Staubli VAL3: SparePoint.pjx

--- SparePoint.pjx ---
Parameters version=s7.8.3 stackSize=5000 millimeterUnit=true
Program file=EditPoint.pgx
Program file=EnterPageKey.pgx
Program file=getPoint.pgx
Program file=Init.pgx
Program file=Main.pgx
Program file=MainKey.pgx
Program file=OnF1.pgx
Program file=OnF2.pgx
Program file=OnF3.pgx
Program file=OnF4.pgx
Program file=OnF5.pgx
Program file=OnF6.pgx
Program file=OnF7.pgx
Program file=OnF8.pgx
Program file=Refresh.pgx
Program file=Refresh2.pgx
Program file=Refresh3.pgx
Program file=RefreshList.pgx
Program file=Save.pgx
Program file=setPoint.pgx
Program file=start.pgx
Program file=stop.pgx
Data file=SparePoint.dtx
Library alias=user path=Disk://userPage/USERPAGE.pjx
Library alias=PublicProg path=Disk://PublicProg/PublicProg.pjx

--- SparePoint.dtx ---
bool bByPass[4]
bool bExit
bool bListRefresh
bool bUserRefresh
frame fFrame = {fatherId=world[0]}
mdesc mNomSpeed
num nPage = 1
num nSelected
public pointRx pPoint{}
  [P1] = {x=495.660657, y=122.165524, z=84.338304, rx=9.53283, ry=179.762496, rz=-66.438432, shoulder=lefty, elbow=epositive, wrist=wpositive, fatherId=world[0]}
  [P10] = {fatherId=world[0]}
  [P11] = {fatherId=world[0]}
  [P12] = {fatherId=world[0]}
  [P13] = {fatherId=world[0]}
  [P14] = {fatherId=world[0]}
  [P15] = {fatherId=world[0]}
  [P16] = {fatherId=world[0]}
  [P2] = {fatherId=world[0]}
  [P3] = {fatherId=world[0]}
  [P4] = {fatherId=world[0]}
  [P5] = {fatherId=world[0]}
  [P6] = {fatherId=world[0]}
  [P7] = {fatherId=world[0]}
  [P8] = {fatherId=world[0]}
  [P9] = {fatherId=world[0]}
public string sDeli[2]
  [0] = "A"
  [1] = "C"
public string sFileList = "A140"
string sFolder = "Disk://Traj/"
string sItem = "P1"
string sList[16]
  [0] = "P1"
  [1] = "P2"
  [2] = "P3"
  [3] = "P4"
  [4] = "P5"
  [5] = "P6"
  [6] = "P7"
  [7] = "P8"
  [8] = "P9"
  [9] = "P10"
  [10] = "P11"
  [11] = "P12"
  [12] = "P13"
  [13] = "P14"
  [14] = "P15"
  [15] = "P16"
string sListItemValue
string sOutputFolder = "Disk://Traj/"
string sParameter
string sPointName = "P1"
string sPtPara

--- Main.pgx ---
program Main()
  local num l_nKey
begin
  //
  do
    call Refresh()
    call RefreshList()
    call user:setList("路径",sList,bUserRefresh,bListRefresh,nSelected,sItem,l_nKey)
    bUserRefresh=false
    bListRefresh=false
    call MainKey(l_nKey)
    delay(0)
  until bExit

end

--- EditPoint.pgx ---
program EditPoint()
  local bool l_bRes
  local num l_i
  local string l_sValue
  local num l_nSelect
  local string l_sItem
  local num l_nKey
  local num l_nRes
begin
//  switch nPage
//    //运动点
//    case 1
//      cls()
//      resize(sParameter,1,11)
//      sParameter[0]="X"
//      sParameter[1]="Y"
//      sParameter[2]="Z"
//      sParameter[3]="Rx"
//      sParameter[4]="Ry"
//      sParameter[5]="Rz"
//      sParameter[6]="P1"
//      sParameter[7]="P2"
//      sParameter[8]="IO1"
//      sParameter[9]="IO2"
//      sParameter[10]="delay"
//      //
//      resize(sListItemValue,1,size(sParameter))
//      sListItemValue[0]=toString(".3",prd:pDemo[nSelected].trsf.x)
//      sListItemValue[1]=toString(".3",prd:pDemo[nSelected].trsf.y)
//      sListItemValue[2]=toString(".3",prd:pDemo[nSelected].trsf.z)
//      sListItemValue[3]=toString(".3",prd:pDemo[nSelected].trsf.rx)
//      sListItemValue[4]=toString(".3",prd:pDemo[nSelected].trsf.ry)
//      sListItemValue[5]=toString(".3",prd:pDemo[nSelected].trsf.rz)
//      //解析sPtParameter
//      call getPtPara(prd:sPtParameter[nSelected],sPtPara)
//      sListItemValue[6]=sPtPara[0]
//      sListItemValue[7]=sPtPara[1]
//      sListItemValue[8]=sPtPara[2]
//      sListItemValue[9]=sPtPara[3]
//      sListItemValue[10]=sPtPara[4]
//      //
//      for l_i=0 to size(sParameter)-1
//        call user:strlength(sParameter[l_i],user:nBottomX/2)
//        l_sValue=sListItemValue[l_i]
//        call user:strlength(l_sValue,user:nBottomX/2+1)
//        sParameter[l_i]=sParameter[l_i]+":"+l_sValue
//      endFor

//      bUserRefresh=true
//      bListRefresh=true
//      //
//      do
//        if bUserRefresh
//          cls()
//          call user:clear(0,13)
//          call user:typeMenu(8,"确定")
//        endIf
//        call user:setList("编辑点",sParameter,bUserRefresh,bListRefresh,l_nSelect,l_sItem,l_nKey)
//        bUserRefresh=false
//        bListRefresh=false
//        call EnterPageKey(l_nKey,l_nSelect,sParameter[l_nSelect])
//        delay(0)
//      until l_nKey==255 or l_nKey==278
//      prd:sPtParameter[nSelected]=sListItemValue[6]+"/"+sListItemValue[7]+"/"+sListItemValue[8]+"/"+sListItemValue[9]+"/"+sListItemValue[10]
//      bUserRefresh=true
//      bListRefresh=true
//    break
//  endSwitch
end

--- EnterPageKey.pgx ---
program EnterPageKey(num& x_nKey, num& x_nSelect, string& x_sItem)
  local string l_sStr
  local num l_nKey
  local string l_sEmpty
  local string l_sValue
  local num l_nItem
  local num l_nView
  local string l_sItem
  local point lp
  local string l_sYN[2]
  local bool l_bRes
  local num l_nTemp
begin
  //
//  //编辑项目
//  switch x_nSelect
//    //X
//    case 0
//      if x_nKey==270
//        call user:editNum(x_sItem,sListItemValue[x_nSelect],prd:pDemo[nSelected].trsf.x,x_nSelect)
//      endIf
//    break
//    //Y
//    case 1
//      if x_nKey==270
//        call user:editNum(x_sItem,sListItemValue[x_nSelect],prd:pDemo[nSelected].trsf.y,x_nSelect)
//      endIf
//    break
//    //Z
//    case 2
//      if x_nKey==270
//        call user:editNum(x_sItem,sListItemValue[x_nSelect],prd:pDemo[nSelected].trsf.z,x_nSelect)
//      endIf
//    break
//    //rx
//    case 3
//      if x_nKey==270
//        call user:editNum(x_sItem,sListItemValue[x_nSelect],prd:pDemo[nSelected].trsf.rx,x_nSelect)
//      endIf
//    break
//    //ry
//    case 4
//      if x_nKey==270
//        call user:editNum(x_sItem,sListItemValue[x_nSelect],prd:pDemo[nSelected].trsf.ry,x_nSelect)
//      endIf
//    break
//    //rz
//    case 5
//      if x_nKey==270
//        call user:editNum(x_sItem,sListItemValue[x_nSelect],prd:pDemo[nSelected].trsf.rz,x_nSelect)
//      endIf
//    break
//    //P1
//    case 6
//      if x_nKey==270
//        // call user:editNum(x_sItem,sListItemValue[x_nSelect],Path:mTrajSpd[nSelectedC].tvel,x_nSelect)
//      endIf
//    break
//    //P2
//    case 7
//      if x_nKey==270
//        //call user:editNum(x_sItem,sListItemValue[x_nSelect],Path:mTrajSpd[nSelectedC].accel,x_nSelect)
//      endIf
//    break
//    //IO1
//    case 8
//      if x_nKey==270
//        call IO:setIO(sListItemValue[x_nSelect])
//        call IO:Main(1)
//        call IO:getIO(sListItemValue[x_nSelect])
//        //
//        x_sItem="IO1      :"+sListItemValue[x_nSelect]
//      endIf

//    break
//    //IO2
//    case 9
//      if x_nKey==270
//        call IO:setIO(sListItemValue[x_nSelect])
//        call IO:Main(1)
//        call IO:getIO(sListItemValue[x_nSelect])
//        //
//        x_sItem="IO2      :"+sListItemValue[x_nSelect]
//      endIf
//    break
//    //delay
//    case 10
//      if x_nKey==270
//        call user:editNum(x_sItem,sListItemValue[x_nSelect],l_nTemp,x_nSelect)
//      endIf
//    break
//  endSwitch
//  if x_nKey==270
//    bUserRefresh=true
//    bListRefresh=true
//  endIf
end

--- getPoint.pgx ---
public program getPoint(string& x_sPoint)
begin
  //
  x_sPoint=sPointName
end

--- Init.pgx ---
program Init()
  local num l_ni
begin
  //
  bUserRefresh=bListRefresh=true
  //
  bExit=false

end

--- MainKey.pgx ---
program MainKey(num x_nKey)
  local num l_nKey
begin
  //
  switch x_nKey
    //记录
    case 271
      call OnF1()
    break
    //
    case 272
      call OnF2()
    break
    //
    case 273
      call OnF3()
    break
    //
    case 274
      call OnF4()
    break
    //
    case 275
    break
    //
    case 276
      call OnF6()
    break
    //save
    case 277
      call OnF7()
    break
    //返回
    case 278
      call OnF8("是否返回")
    break
    case 270
      call EditPoint()
    break
  endSwitch
end

--- OnF1.pgx ---
program OnF1()
  local bool l_bRes
begin

  pPoint[sItem]=here(flange,world)

end

--- OnF2.pgx ---
program OnF2()
  local num l_ni
  local bool l_bRes
begin

  call setPoint(sItem)
  popUpMsg("选择点："+sItem)
end

--- OnF3.pgx ---
program OnF3()
begin

end

--- OnF4.pgx ---
program OnF4()
  local string l_sProperty[2]
  local string l_sItem
begin
//  //调用tool or frame library
//  l_sProperty[0]="工具"
//  l_sProperty[1]="坐标系"
//  call user:SetProerty("",26,9,6,2,l_sProperty,l_sItem)
//  if l_sItem=="工具"
//    call Tool:setTool(prd:sToolName)
//    call Tool:Main(1)
//    call Tool:getTool(prd:sToolName)
//  elseIf l_sItem=="坐标系"
//    call Frame:SetFrame(prd:sFrameName)
//    call Frame:Main(1)
//    call Frame:getFrame(prd:sFrameName)
//  endIf
//  bUserRefresh=bListRefresh=true
end

--- Refresh.pgx ---
program Refresh()
begin
  //编辑界面
  if bUserRefresh
    cls()
    userPage()
    gotoxy(1,1)
    put("F1->记录")
    gotoxy(1,13)
    put("F1")
    gotoxy(1,2)
    put("F2->确定")
    gotoxy(6,13)
    put("F2")
//    gotoxy(1,3)
//    put("F3->删除")
//    gotoxy(11,13)
//    put("F3")
//    gotoxy(1,4)
//    put("F4->选择工具/坐标系")
//    gotoxy(16,13)
//    put("F4")

//    gotoxy(1,5)
//    put("F5->运动方向切换")
//    gotoxy(21,13)
//    put("F5")
    //    gotoxy(1,6)
    //    put("F6->")
    //    gotoxy(26,13)
    //    put("")
    gotoxy(1,7)
    put("F7->保存")
    gotoxy(31,13)
    put("F7")
    gotoxy(1,8)
    put("F8->返回")
    gotoxy(36,13)
    put("F8")

  endIf
end

--- Refresh2.pgx ---
program Refresh2()
begin
  //模拟界面
  if bUserRefresh
    cls()
    userPage()
    gotoxy(1,1)
    put("F1->开始/继续")
    gotoxy(1,13)
    put("F1")
    gotoxy(1,2)
    put("F2->停止")
    gotoxy(6,13)
    put("F2")
//    gotoxy(1,3)
//    put("F3->删除")
//    gotoxy(11,13)
//    put("F3")
//    gotoxy(1,4)
//    put("F4->选择工具/坐标系")
//    gotoxy(16,13)
//    put("F4")
    //
//    gotoxy(1,6)
//    put("F6->")
//    gotoxy(26,13)
//    put("")
//    gotoxy(1,7)
//    put("F7->保存")
//    gotoxy(31,13)
//    put("F7")
    gotoxy(1,8)
    put("F8->返回")
    gotoxy(36,13)
    put("F8")
  endIf
end

--- RefreshList.pgx ---
program RefreshList()
  local num l_ni
begin
  if bListRefresh
    resize(sList,1,size(pPoint))
    for l_ni=0 to size(pPoint)-1
      sList[l_ni]="P"+toString("",l_ni+1)
    endFor
  endIf
end

--- Save.pgx ---
program Save()
  local num l_ni
begin
  //
  libSave()
  popUpMsg("保存完毕!")
end

--- setPoint.pgx ---
public program setPoint(string x_sPoint)
begin
  //
  sPointName=x_sPoint
end
